// TIA Portal V17 export
// export: Created 2025-03-10T13:12:13.9149476Z, ExportSetting WithDefaults, DisplayName Totally Integrated Automation Portal, DisplayVersion V17 Update 8, DisplayName TIA Portal Openness, DisplayVersion V17 Update 8, DisplayName TIA Portal Version Control Interface, DisplayVersion V17, DisplayName SINAMICS Startdrive Advanced, DisplayVersion V17 SP2, DisplayName SINAMICS Startdrive G110M, G120, G120C, G120D, G120P, G115D, DisplayVersion V17 SP2, DisplayName SINAMICS Startdrive G130, G150, S120, S150, SINAMICS MV, S210, DisplayVersion V17 SP2, DisplayName STEP 7 Professional, DisplayVersion V17 Update 8, DisplayName SINUMERIK ONE STEP 7 Toolbox, DisplayVersion V17 Update 12, DisplayName SINUMERIK 840D sl STEP 7 Toolbox, DisplayVersion V17 Update 12, DisplayName STEP 7 Safety, DisplayVersion V17 Update 6, DisplayName WinCC Advanced, DisplayVersion V17 Update 8
TYPE "SMC_JXCP1_TO_PLC"
// stored: IsFailsafeCompliant false
   STRUCT
      STEP_NUMBER_OUT_0 : Bool := false;   // STEP NUMBER BINARY DIGIT 0
      STEP_NUMBER_OUT_1 : Bool := false;   // STEP NUMBER BINARY DIGIT 1
      STEP_NUMBER_OUT_2 : Bool := false;   // STEP NUMBER BINARY DIGIT 2
      STEP_NUMBER_OUT_3 : Bool := false;   // STEP NUMBER BINARY DIGIT 3
      STEP_NUMBER_OUT_4 : Bool := false;   // STEP NUMBER BINARY DIGIT 4
      STEP_NUMBER_OUT_5 : Bool := false;   // STEP NUMBER BINARY DIGIT 5
      STEP_NUMBER_UNUSED_6 : Bool := false;   // -
      STEP_NUMBER_UNUSED_7 : Bool := false;   // -
      BUSY : Bool;   // CONTROLLER BUSY (MOVEMENT)
      SVRE : Bool;   // SERVO MOTOR STATUS (ON/OFF)
      STON : Bool;   // POSITION INFORMATION/STATUS ESTABLISHED
      INP : Bool;   // IN POSITION
      AREA : Bool;   // BETWEEN AREA 1 AND AREA 2 IN STEP DATA
      WAREA : Bool;   // BETWEEN W AREA 1 AND W AREA 2 IN STEP DATA
      ESTOP : Bool;   // TEACHING BOX EMERGENCY STOP
      ALARM : Bool;   // ALARM PRESENT
      UNUSED_2_0 : Bool;   // -
      UNUSED_2_1 : Bool;   // -
      UNUSED_2_2 : Bool;   // -
      UNUSED_2_3 : Bool;   // -
      READY : Bool;   // SERVO ON AND NO ALARMS
      UNUSED_2_5 : Bool;   // -
      UNUSED_2_6 : Bool;   // -
      UNUSED_2_7 : Bool;   // -
      UNSUSED_3_0 : Bool;   // -
      UNSUSED_3_1 : Bool;   // -
      UNSUSED_3_2 : Bool;   // -
      UNSUSED_3_3 : Bool;   // -
      UNSUSED_3_4 : Bool;   // -
      UNSUSED_3_5 : Bool;   // -
      UNSUSED_3_6 : Bool;   // -
      UNSUSED_3_7 : Bool;   // -
      CURRENT_POSITION : DWord;   // CURRENT ACTUATOR POSITION (MULTIPLES OF 0.01mm)
      CURRENT_SPEED : Word;   // CURRENT ACTUATOR SPEED (MULTIPLES OF 1mm/s)
      CURRENT_PUSHING_FORCE : Word;   // CURRENT ACTUATOR PUSHING FORCE (MULTIPLES OF 1%)
      TARGET_POSITION : DWord;   // TARGET ACTUATOR POSITION (MULTIPLES OF 0.01mm)
      ALARM_1 : DWord;   // ALARM 1 CODE
      ALARM_2 : DWord;   // ALARM 2 CODE
      ALARM_3 : DWord;   // ALARM 3 CODE
      ALARM_4 : DWord;   // ALARM 4 CODE
   END_STRUCT;
END_TYPE
